{attribute 'GeneratedUsingTerminal: EL3681-0000-0017'}
{attribute addProperty BoxType "EL3681-0000-0017"}
{attribute addProperty Id "ModeBYTE1RangeSINT1"}
{attribute addProperty CRC "616581440"}
{attribute addProperty Size "2"}
TYPE Setting_24C04940 :
STRUCT
	{attribute addProperty Name "Mode"}
	Mode : BYTE;
	{attribute addProperty Name "Range"}
	Range : SINT;
END_STRUCT
END_TYPE

(* stored: Version 1.2.0.0, ProductVersion 3.1.4024.9
   DUT Setting_24C04940: Id {ef666ee6-0633-4791-b27e-56a14c1b9e94} *)
